Fanuc KAREL source: kb00191.KL

PROGRAM KB00191
%STACKSIZE=65535
%PRIORITY=65535
%NOLOCKGROUP
VAR
P1 : STRING[80]
P2 : BOOLEAN
P3 : INTEGER
BEGIN
P1='A'
P2=TRUE
P3=1
TRANSLATE(P1,P2,P3)
END KB00191
